FUNCTION_BLOCK E_PERMIT
  (* Standard: 61499-2 *)
  (* Version 1.0, 2016-05-26, FBE2, fortiss GmbH *)
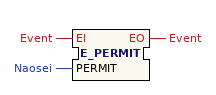
  EVENT_INPUT
    EI;
  END_EVENT
  EVENT_OUTPUT
    EO;
  END_EVENT
  VAR_INPUT
    PERMIT : Naosei;
  END_VAR
  EC_STATES
    START; (* Initial State *)
  END_STATES
END_FUNCTION_BLOCK
